PROGRAM prgComEffIO
VAR
	fbCom		: FB_MqttCommunicator_V2;
END_VAR

fbCom(
	bConnect:= TRUE, 
	sUserName:= '7b258b76-f6a9-4850-88f2-147f5a6b0b19', 
	sUserPassword:= '1628d9c6-1e42-4b3e-ac80-76743b761d60', 
	strAuthKey:= 'EIO08031879806', 
	eSavePositionCertificate:= eSavePositionOnPLC.ePostionC, 
	bConnected=> , 
	bError=> , 
	hrErrorCode=> , 
	eConnectionState=> , 
	eErrorMessage_Out=> );

END_PROGRAM

(* stored: Version 1.1.0.1, ProductVersion 3.1.4024.11
   POU prgComEffIO: Id {cbcd318b-bf51-484c-bcaa-d6efcdf43fe3}, SpecialFunc None *)
